Yaskawa INFORM job: REF_DETAL.JBI

/JOB
//NAME REF_DETAL
///FOLDERNAME INNE
//POS
///NPOS 3,3,0,0,0,0
///TOOL 0
///POSTYPE PULSE
///PULSE
C00000=-100501,-66055,-20899,-62068,82879,-39866
C00001=-152051,96304,51052,-64402,59757,50959
C00002=234348,-79836,-91898,-37770,17442,-34800
BC00000=363518,7679,447953
BC00001=363518,7678,856292
BC00002=363518,7678,856290
//INST
///DATE 2023/10/17 17:52
///ATTR SC,RW
///GROUP1 RB1,BS1
NOP
MOVJ C00000 BC00000 VJ=10.00 PL=0
MOVJ C00001 BC00001 VJ=0.78 PL=0
MOVJ C00002 BC00002 VJ=0.78 PL=0
END
